FUNCTION_BLOCK RESET_BTNs (* Composite Function Block Type *)
  (* Standard: 61499-2 *)
  (* Version 0.0, 6/18/2026, Schneider Electric, template *)
  PACKAGE SE.Nereda;
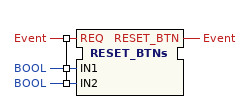
  EVENT_INPUT
    REQ WITH IN1, IN2; (* Normal Execution Request *)
  END_EVENT
  EVENT_OUTPUT
    RESET_BTN;
  END_EVENT
  VAR_INPUT
    IN1 : BOOL; (* Argument *)
    IN2 : BOOL; (* Argument *)
  END_VAR
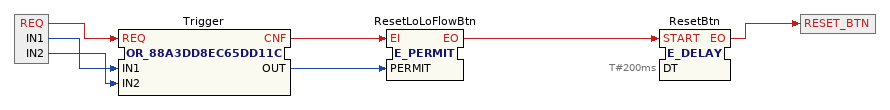
  FBS
    ResetBtn : E_DELAY(DT := T#200ms);
    ResetLoLoFlowBtn : E_PERMIT;
    Trigger : OR_88A3DD8EC65DD11C; {SET_ATTRIBUTE(Configuration.GenericFBType.InterfaceParams, Runtime.Standard#CNT:=2;OUT:BOOL)}
  END_FBS
  EVENT_CONNECTIONS
    ResetBtn.EO TO RESET_BTN;
    ResetLoLoFlowBtn.EO TO ResetBtn.START;
    Trigger.CNF TO ResetLoLoFlowBtn.EI;
    REQ TO Trigger.REQ;
  END_CONNECTIONS
  DATA_CONNECTIONS
    Trigger.OUT TO ResetLoLoFlowBtn.PERMIT;
    IN1 TO Trigger.IN1;
    IN2 TO Trigger.IN2;
  END_CONNECTIONS
END_FUNCTION_BLOCK
